FUNCTION_BLOCK TwoConCtlMulti (* Composite Function Block Type *)
  (* Standard: 61499-2 *)
  (* Version 0.2, 2003-12-05, JHC, Rockwell Automation, Renamed from NEWCOMPFB. *)
  (* Version 0.1, 2002-01-08, JHC, Rockwell Automation, Added DLY FB as example. *)
  (* Version 0.0, 2000-05-27, JHC, Rockwell Automation *)
  (* Compiler header: package fb.rt.conveyorIEC61499; *)
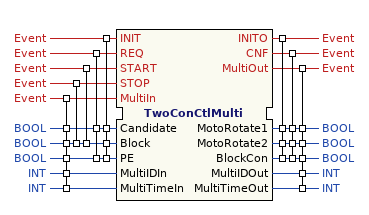
  EVENT_INPUT
    INIT WITH Candidate, Block, PE; (* Initialization Request *)
    REQ WITH Candidate, PE; (* Normal Execution Request *)
    START WITH Block;
    STOP WITH Block;
    MultiIn WITH Candidate, Block, PE, MultiIDIn, MultiTimeIn; (* Multicast Input Event *)
  END_EVENT
  EVENT_OUTPUT
    INITO WITH MotoRotate1, MotoRotate2, BlockCon; (* Initialization Confirm *)
    CNF WITH MotoRotate1, MotoRotate2, BlockCon; (* Execution Confirmation *)
    MultiOut WITH MultiIDOut, MotoRotate1, MotoRotate2, BlockCon, MultiTimeOut; (* Multicast Output Event *)
  END_EVENT
  VAR_INPUT
    Candidate : BOOL;
    Block : BOOL;
    PE : BOOL;
    MultiIDIn : INT;
    MultiTimeIn : INT;
  END_VAR
  VAR_OUTPUT
    MotoRotate1 : BOOL;
    MotoRotate2 : BOOL;
    BlockCon : BOOL;
    MultiIDOut : INT;
    MultiTimeOut : INT;
  END_VAR
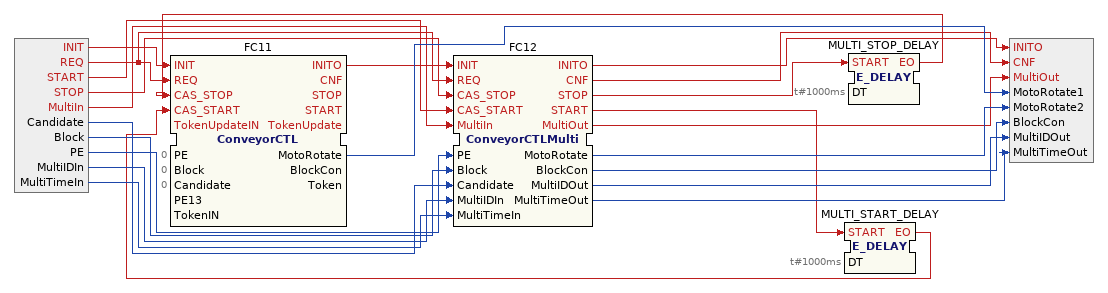
  FBS
    FC11 : ConveyorCTL(PE := 0, Block := 0, Candidate := 0);
    FC12 : ConveyorCTLMulti;
    MULTI_STOP_DELAY : E_DELAY(DT := t#1000ms);
    MULTI_START_DELAY : E_DELAY(DT := t#1000ms);
  END_FBS
  EVENT_CONNECTIONS
    INIT TO FC11.INIT;
    REQ TO FC11.REQ;
    FC12.INITO TO INITO;
    FC12.CNF TO CNF;
    REQ TO FC12.REQ;
    STOP TO FC12.CAS_STOP;
    START TO FC12.CAS_START;
    FC11.INITO TO FC12.INIT;
    MultiIn TO FC12.MultiIn;
    FC12.MultiOut TO MultiOut;
    FC12.STOP TO MULTI_STOP_DELAY.START;
    MULTI_STOP_DELAY.EO TO FC11.CAS_STOP;
    FC12.START TO MULTI_START_DELAY.START;
    MULTI_START_DELAY.EO TO FC11.CAS_START;
  END_CONNECTIONS
  DATA_CONNECTIONS
    Block TO FC12.Block;
    Candidate TO FC12.Candidate;
    FC12.BlockCon TO BlockCon;
    FC11.MotoRotate TO MotoRotate1;
    FC12.MotoRotate TO MotoRotate2;
    MultiIDIn TO FC12.MultiIDIn;
    MultiTimeIn TO FC12.MultiTimeIn;
    FC12.MultiIDOut TO MultiIDOut;
    FC12.MultiTimeOut TO MultiTimeOut;
    PE TO FC12.PE;
  END_CONNECTIONS
END_FUNCTION_BLOCK
